INTERFACE IInputDevice EXTENDS IDevice

METHOD UpdateStateFromInputs
END_METHOD

END_INTERFACE

(* stored: Version 1.1.0.1
   Itf IInputDevice: Id {352f94cf-b25f-4229-a5b2-4644d6346715}
   Method UpdateStateFromInputs: Id {9900a606-26fe-4855-94ce-49bffd62a979} *)
